{attribute addProperty BoxType "EL3413-0000-0016"}
{attribute addProperty Id "TxPDO_ToggleBIT10.12516"}
{attribute addProperty CRC "195118718"}
{attribute addProperty SizeInBites "16"}
{attribute addProperty SizeInBytes "2"}
TYPE STATUS_0BA1467E :
STRUCT
	{attribute 'hide'}
	reserve_1_BIT_0 : BIT;
	{attribute 'hide'}
	reserve_1_BIT_1 : BIT;
	{attribute 'hide'}
	reserve_1_BIT_2 : BIT;
	{attribute 'hide'}
	reserve_1_BIT_3 : BIT;
	{attribute 'hide'}
	reserve_1_BIT_4 : BIT;
	{attribute 'hide'}
	reserve_1_BIT_5 : BIT;
	{attribute 'hide'}
	reserve_1_BIT_6 : BIT;
	{attribute 'hide'}
	reserve_1_BIT_7 : BIT;
	{attribute 'hide'}
	reserve_1_BIT_8 : BIT;
	{attribute 'hide'}
	reserve_1_BIT_9 : BIT;
	{attribute 'hide'}
	reserve_1_BIT_10 : BIT;
	{attribute 'hide'}
	reserve_1_BIT_11 : BIT;
	{attribute 'hide'}
	reserve_1_BIT_12 : BIT;
	{attribute 'hide'}
	reserve_1_BIT_13 : BIT;
	{attribute 'hide'}
	reserve_1_BIT_14 : BIT;
	{attribute addProperty Name "TxPDO_Toggle"}
	TxPDO_Toggle : BIT;
END_STRUCT
END_TYPE

(* stored: Version 1.2.0.0, ProductVersion 3.1.4024.9
   DUT STATUS_0BA1467E: Id {1415fe2f-350a-4956-9740-5b479ce76254} *)
